{attribute 'Tc2GvlVarNames'}
VAR_CONFIG
END_VAR

(* stored: Version 1.1.0.1, ProductVersion 3.1.4024.10
   GVL Variable_Configuration: Id {41d0122b-c58e-45ba-96d0-5b271401c99e} *)
